(* IEC 61131-3 sources: Explicit_MPC_on_PLC/Quad-Tank/MATLAB_Files/Used Files/plcsrc (part 2) *)

        (* InitializeConditions for UnitDelay: '<S3>/last_mv' *)
        last_mv_DSTATE[0] := 0.0;
        last_mv_DSTATE[1] := 0.0;
        (* End of SystemInitialize for SubSystem: '<Root>/Explicit Controller' *)
    SS_STEP:
        (* Outputs for Atomic SubSystem: '<Root>/Explicit Controller' *)
        (* MATLAB Function: '<S3>/Explicit MPC Evaluation' *)
        (* MATLAB Function 'Explicit MPC Controller/MPC/Explicit MPC Evaluation': '<S4>:1' *)
        (* '<S4>:1:6' coder.extrinsic('mpcblock_pwa_evaluate_double_mex'); *)
        (* '<S4>:1:7' coder.extrinsic('mpcblock_pwa_evaluate_single_mex'); *)
        (* Parameters *)
        (* '<S4>:1:10' isSimulation = coder.target('Sfun') && ~coder.target('RtwForRapid') && ~coder.target('RtwForSim'); *)
        (* '<S4>:1:11' isDouble = isa(r,'double'); *)
        (* '<S4>:1:12' ZERO = zeros('like',r); *)
        (* '<S4>:1:13' ONE = ones('like',r); *)
        (* Pre-allocate all the MEX block outputs for the simulation mode *)
        (* '<S4>:1:18' if isSimulation *)
        (* '<S4>:1:26' if isSimulation *)
        (* '<S4>:1:39' else *)
        (* When doing code generation, use M code directly *)
        (* '<S4>:1:41' [u, status, region, new_x, xest] = mpcblock_pwa_evaluate(old_x, r, v, ym, ext_u, old_u, no_mv, nu, nx, nv, uoff, ... *)
        (* '<S4>:1:42'         openloopflag, F, G, H, K, i1, i2, nr, np, xunfindex, refunfindex, uunfindex, mdunfindex,thmin,thmax,... *)
        (* '<S4>:1:43'         CustomEstimation, RMYscale, myoff, xoff, A, Bu, Bv, Cm, Dvm, M, L, ... *)
        (* '<S4>:1:44'         switch_in, switch_inport, no_switch, enable_value); *)
        regionmin := 1;
        b_k := -1;
        (* End of Outputs for SubSystem: '<Root>/Explicit Controller' *)
        (* Outputs for Atomic SubSystem: '<Root>/Explicit Controller' *)
        (* MATLAB Function: '<S3>/Explicit MPC Evaluation' incorporates:
         *  Memory: '<S3>/last_x' *)
        FOR i := 0 TO 5 DO
            new_x[i] := last_x_PreviousInput[i];
        END_FOR;
        (* End of Outputs for SubSystem: '<Root>/Explicit Controller' *)
        (* Outputs for Atomic SubSystem: '<Root>/Explicit Controller' *)
        (* MATLAB Function: '<S3>/Explicit MPC Evaluation' *)
        FOR i := 0 TO 1 DO
            betamin := 0.0;
            FOR b_h := 0 TO 5 DO
                betamin := (Explicit_b_Cm[(b_h * 2) + i] * new_x[b_h]) + betamin;
            END_FOR;
            y_innov[i] := MeasuredTankOutputs[i] - betamin;
        END_FOR;
        (* End of Outputs for SubSystem: '<Root>/Explicit Controller' *)
        (* Outputs for Atomic SubSystem: '<Root>/Explicit Controller' *)
        (* MATLAB Function: '<S3>/Explicit MPC Evaluation' *)
        FOR i := 0 TO 5 DO
            rtb_xest[i] := ((Explicit_b_M[i + 6] * y_innov[1]) + (Explicit_b_M[i] * y_innov[0])) + new_x[i];
        END_FOR;
        (* End of Outputs for SubSystem: '<Root>/Explicit Controller' *)
        (* Outputs for Atomic SubSystem: '<Root>/Explicit Controller' *)
        (* MATLAB Function: '<S3>/Explicit MPC Evaluation' incorporates:
         *  UnitDelay: '<S3>/last_mv' *)
        FOR i := 0 TO 9 DO
            th[i] := 0.0;
        END_FOR;
        FOR b_h := 0 TO 5 DO
            th[b_h] := rtb_xest[b_h];
        END_FOR;
        th[6] := ref[0];
        th[8] := last_mv_DSTATE[0];
        th[7] := ref[1];
        th[9] := last_mv_DSTATE[1];
        FOR b_h := 0 TO 9 DO
            betamin := th[b_h];
            IF betamin < Explicit_b_thmin[b_h] THEN
                regionmin := 0;
            ELSIF betamin > Explicit_b_thmax[b_h] THEN
                regionmin := 0;
            END_IF;
        END_FOR;
        du[0] := 0.0;
        du[1] := 0.0;
        IF regionmin = 1 THEN
            found := FALSE;
            regionmin := 0;
            betamin := 1.797693134862316E+307;
            WHILE ( NOT found) AND ((b_k + 1) < 101) DO
                b_k := b_k + 1;
                b_h := INT_TO_DINT(b_i1[b_k]);
                beta := -1.0;
                WHILE b_h <= INT_TO_DINT(b_i2[b_k]) DO
                    betah := 0.0;
                    FOR i := 0 TO 9 DO
                        betah := (Explicit_g_H[((1978 * i) + b_h) - 1] * th[i]) + betah;
                    END_FOR;
                    betah := betah - Explicit_c_K[b_h - 1];
                    IF betah > beta THEN
                        beta := betah;
                    END_IF;
                    b_h := b_h + 1;
                END_WHILE;
                IF beta <= 0.0 THEN
                    found := TRUE;
                ELSIF betamin > beta THEN
                    betamin := beta;
                    regionmin := b_k + 1;
                END_IF;
            END_WHILE;
            IF  NOT found THEN
                b_k := regionmin - 1;
            END_IF;
            b_k := DWORD_TO_DINT(SHL(DINT_TO_DWORD(b_k), 1));
            FOR regionmin := 0 TO 1 DO
                b_h := regionmin + b_k;
                betamin := 0.0;
                FOR i := 0 TO 9 DO
                    betamin := (Explicit_b_F[(202 * i) + b_h] * th[i]) + betamin;
                END_FOR;
                du[regionmin] := Explicit_b_G[regionmin + b_k] + betamin;
            END_FOR;
        END_IF;
        betamin := last_mv_DSTATE[0] + du[0];
        beta := betamin;
        mv[0] := betamin;
        betamin := last_mv_DSTATE[1] + du[1];
        (* End of Outputs for SubSystem: '<Root>/Explicit Controller' *)
        (* Outputs for Atomic SubSystem: '<Root>/Explicit Controller' *)
        FOR i := 0 TO 5 DO
            (* MATLAB Function: '<S3>/Explicit MPC Evaluation' *)
            rtb_xest[i] := 0.0;
            FOR b_h := 0 TO 5 DO
                rtb_xest[i] := (Explicit_b_A[(6 * b_h) + i] * new_x[b_h]) + rtb_xest[i];
            END_FOR;
            (* Update for Memory: '<S3>/last_x' incorporates:
             *  MATLAB Function: '<S3>/Explicit MPC Evaluation' *)
            last_x_PreviousInput[i] := ((Explicit_b_L[i + 6] * y_innov[1]) + (Explicit_b_L[i] * y_innov[0])) + (rtb_xest[i] + ((Explicit_b_Bu[i + 6] * betamin) + (Explicit_b_Bu[i] * beta)));
        END_FOR;
        (* Update for UnitDelay: '<S3>/last_mv' *)
        last_mv_DSTATE[0] := mv[0];
        (* Outport: '<Root>/mv' incorporates:
         *  Gain: '<S3>/ext.mv_scale1'
         *  UnitDelay: '<S3>/last_mv' *)
        mv[0] := 0.15299877600979192 * mv[0];
        (* Update for UnitDelay: '<S3>/last_mv' *)
        last_mv_DSTATE[1] := betamin;
        (* Outport: '<Root>/mv' incorporates:
         *  Gain: '<S3>/ext.mv_scale1' *)
        mv[1] := 0.15299877600979192 * betamin;
        (* End of Outputs for SubSystem: '<Root>/Explicit Controller' *)
END_CASE;
END_FUNCTION_BLOCK
VAR_GLOBAL CONSTANT
    SS_INITIALIZE: SINT := 0;
    SS_STEP: SINT := 1;
END_VAR
